Universal Robots PolyScope program: Cinta_1.urp

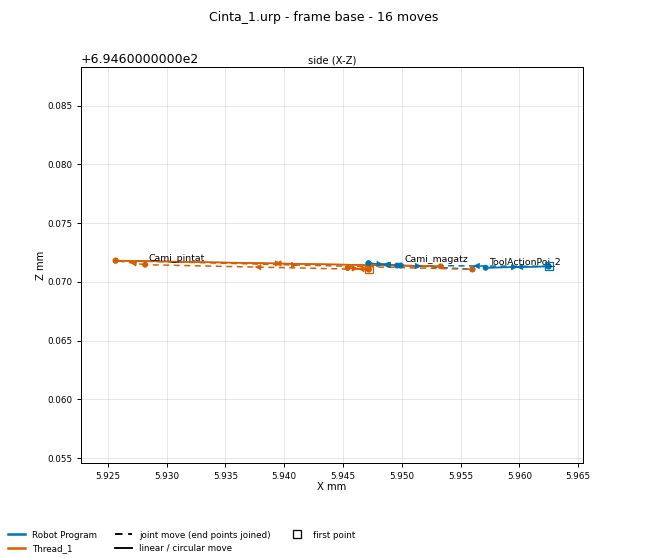
[picture p0: tool path of Cinta_1.urp in frame base, 16 of 16 moves have a stored position in this frame; points joined in program order, loops and branches not executed]
Program Cinta_1 (installation=default directory=/programs createdIn=5.14.5 lastSavedIn=5.14.5 robotSerialNumber=20195300809)
Calibrated DH parameters: a=[-0.000085, -0.20076, -0.212369, 0.000121, -0.000118, 0]; d=[0.15185, -26.306375, 24.753047, 1.684739, 0.085386, 0.092088]; alpha=[1.572149, -0.00522, -0.011864, 1.571339, -1.571085, 0]; deltaTheta=[0, 0.599885, -0.513355, -0.086555, 0.000006, 0]
InitVariablesNode variables(variable(name=Pallet_1_cnt_1, expression=1), variable(name=Pallet_1_lct, expression=1), variable(name=Pallet_1_lno, expression=1), variable(name=Pallet_1_sep, expression=False), variable(name=Pallet_1_tct, expression=1), variable(name=Pallet_2_cnt_1, expression=1), variable(name=Pallet_2_lct, expression=1), variable(name=Pallet_2_lno, expression=1), variable(name=Pallet_2_sep, expression=False), variable(name=Pallet_2_tct, expression=1), variable(name=Pallet_3_cnt, expression=1), variable(name=Pallet_3_lct, expression=1), variable(name=Pallet_3_lno, expression=1), variable(name=Pallet_3_sep, expression=False), variable(name=Pallet_3_tct, expression=1), variable(name=Pallet_4_cnt, expression=1), variable(name=Pallet_4_lct, expression=1), variable(name=Pallet_4_lno, expression=1), variable(name=Pallet_4_sep, expression=False), variable(name=Pallet_4_tct, expression=1))
Robot Program (runOnlyOnce=false)
  If timer_1≟5  and inici≟get_actual_tcp_pose()
    URCap Palletizing (polyscope-pallet-impl, Universal Robots) dataModel(palletFeature=Base, isPalletizing=false, Variable(key=name, variable(name=Pallet_3)), Variable(key=globalCountingVariable, variable(name=Pallet_3_cnt, initializeExpression=1)), Variable(key=layerNumberVariable, variable(name=Pallet_3_lno, initializeExpression=1)), Variable(key=layerCountingVariable, variable(name=Pallet_3_lct, initializeExpression=1)), Variable(key=handleSeparatorVariable, variable(name=Pallet_3_sep, initializeExpression=False)), Variable(key=totalCountVariable, variable(name=Pallet_3_tct, initializeExpression=1)), Length(key=objectHeight value=0.05 unit=M), Variable(key=referencePoint, variable(featureName=referencePoin_2)), Variable(key=separatorPoint, variable(featureName=separatorPoin_2))); state(isChildrenLocked=true)
      URCap Patterns (polyscope-pallet-impl, Universal Robots) state(isChildrenLocked=true)
        URCap Pattern (polyscope-pallet-impl, Universal Robots) dataModel(UUID=57716a2e-ea0b-4b86-9d22-23fb6d1bb1b5, patternType=IRREGULAR, Variable(key=nameVariable, variable(name=Irreg_Pattern_3))); state(isChildrenLocked=true)
          URCap Item (polyscope-pallet-impl, Universal Robots) dataModel(UUID=925eac26-10bc-4873-a4ec-01d33931e9e1, patternType=IRREGULAR, index=0, calibrationDeltaTheta=[2.0871938292282843E-8, 0.5998849625986696, -0.513354759222901, -0.08655474087847535, 6.239817607139875E-6, -6.658617090343766E-8], calibrationA=[-8.52060452638757E-5, -0.2007601879611388, -0.2123691625519033, 1.2105607098011576E-4, -1.1833705743435544E-4, 0.0], calibrationD=[0.15184970286177432, -26.306374840159272, 24.75304670983349, 1.6847390881089916, 0.085385969004481, 0.09208826337351553], calibrationAlpha=[1.5721487795181908, -0.005219907129425837, -0.011864150755780208, 1.5713392161993658, -1.5710853432049288, 0.0], calibrationJointChecksum=[-1860213401, -1859864814, -1494669377, -1328152407, -1329437658, -1329056899], calibrationStatus=2, calibrationValidChecksum=true, baseToFeature=[0.0, 0.0, 0.0, 0.0, 0.0, 0.0], TCPOffset=[-3.816685185402386E-6, 1.2180760577962246E-7, 0.15000008227769798, -3.269188807254424E-7, 6.278455909932198E-6, -1.926188929202367E-5], Variable(key=variable, variable(name=Item_3)), JointPositions(key=jointpositions, JointPosition(key=[1], Angle(key=pos value=0.000066 unit=RAD)), JointPosition(key=[2], Angle(key=pos value=-1.570806 unit=RAD)), JointPosition(key=[3], Angle(key=pos value=0.000024 unit=RAD)), JointPosition(key=[4], Angle(key=pos value=-1.570762 unit=RAD)), JointPosition(key=[5], Angle(key=pos value=-0.000043 unit=RAD)), JointPosition(key=[6], Angle(key=pos value=-0.000104 unit=RAD))))
      URCap Layers (polyscope-pallet-impl, Universal Robots) dataModel(separators=[false], selectedPatterns=[57716a2e-ea0b-4b86-9d22-23fb6d1bb1b5])
      URCap At Each Item (polyscope-pallet-impl, Universal Robots) dataModel(selectedPattern=57716a2e-ea0b-4b86-9d22-23fb6d1bb1b5, selectedPosition=925eac26-10bc-4873-a4ec-01d33931e9e1, Approach_calibrationDeltaTheta=[2.0871938292282843E-8, 0.5998849625986696, -0.513354759222901, -0.08655474087847535, 6.239817607139875E-6, -6.658617090343766E-8], Approach_calibrationA=[-8.52060452638757E-5, -0.2007601879611388, -0.2123691625519033, 1.2105607098011576E-4, -1.1833705743435544E-4, 0.0], Approach_calibrationD=[0.15184970286177432, -26.306374840159272, 24.75304670983349, 1.6847390881089916, 0.085385969004481, 0.09208826337351553], Approach_calibrationAlpha=[1.5721487795181908, -0.005219907129425837, -0.011864150755780208, 1.5713392161993658, -1.5710853432049288, 0.0], Approach_calibrationJointChecksum=[-1860213401, -1859864814, -1494669377, -1328152407, -1329437658, -1329056899], Approach_calibrationStatus=2, Approach_calibrationValidChecksum=true, Approach_baseToFeature=[0.0, 0.0, 0.0, 0.0, 0.0, 0.0], Approach_TCPOffset=[-9.173349571223492E-6, 4.750605908654393E-9, 0.15000004581161422, -1.2312542340189748E-8, -2.3772295653205082E-5, -6.665466225263506E-6], Exit_calibrationDeltaTheta=[2.0871938292282843E-8, 0.5998849625986696, -0.513354759222901, -0.08655474087847535, 6.239817607139875E-6, -6.658617090343766E-8], Exit_calibrationA=[-8.52060452638757E-5, -0.2007601879611388, -0.2123691625519033, 1.2105607098011576E-4, -1.1833705743435544E-4, 0.0], Exit_calibrationD=[0.15184970286177432, -26.306374840159272, 24.75304670983349, 1.6847390881089916, 0.085385969004481, 0.09208826337351553], Exit_calibrationAlpha=[1.5721487795181908, -0.005219907129425837, -0.011864150755780208, 1.5713392161993658, -1.5710853432049288, 0.0], Exit_calibrationJointChecksum=[-1860213401, -1859864814, -1494669377, -1328152407, -1329437658, -1329056899], Exit_calibrationStatus=2, Exit_calibrationValidChecksum=true, Exit_baseToFeature=[0.0, 0.0, 0.0, 0.0, 0.0, 0.0], Exit_TCPOffset=[1.4942311595496577E-5, 5.093315802451315E-8, 0.1500000438837152, -1.396915314811311E-7, 7.536789619608266E-5, -3.90601478415621E-5], currentWizardState=LANDING, Pose(key=refBaseToFeature, Position(key=posePosition, Length(key=X value=0 unit=M), Length(key=Y value=0 unit=M), Length(key=Z value=0 unit=M)), Rotation(key=poseRotation, Angle(key=RX value=0 unit=RAD), Angle(key=RY value=0 unit=RAD), Angle(key=RZ value=0 unit=RAD))), Pose(key=refPose, Position(key=posePosition, Length(key=X value=0.005957 unit=M), Length(key=Y value=-0.3727 unit=M), Length(key=Z value=0.694671 unit=M)), Rotation(key=poseRotation, Angle(key=RX value=-0.017988 unit=RAD), Angle(key=RY value=2.210197 unit=RAD), Angle(key=RZ value=-2.216559 unit=RAD))), JointPositions(key=Approach_jointpositions, JointPosition(key=[1], Angle(key=pos value=0.000066 unit=RAD)), JointPosition(key=[2], Angle(key=pos value=-1.570806 unit=RAD)), JointPosition(key=[3], Angle(key=pos value=0.000024 unit=RAD)), JointPosition(key=[4], Angle(key=pos value=-1.570762 unit=RAD)), JointPosition(key=[5], Angle(key=pos value=-0.000043 unit=RAD)), JointPosition(key=[6], Angle(key=pos value=-0.000104 unit=RAD))), JointPositions(key=Exit_jointpositions, JointPosition(key=[1], Angle(key=pos value=0.000066 unit=RAD)), JointPosition(key=[2], Angle(key=pos value=-1.570806 unit=RAD)), JointPosition(key=[3], Angle(key=pos value=0.000024 unit=RAD)), JointPosition(key=[4], Angle(key=pos value=-1.570762 unit=RAD)), JointPosition(key=[5], Angle(key=pos value=-0.000043 unit=RAD)), JointPosition(key=[6], Angle(key=pos value=-0.000104 unit=RAD))))
        URCap Generated Movements (polyscope-pallet-impl, Universal Robots) state(isChildrenLocked=true)
          MoveJ speed 60 deg/s, acceleration 80 deg/s^2 (useActiveTCP=true) feature=referencePoin_2
            Waypoint Approach_3: TCP in base x=5.962 y=-372.7 z=694.671 mm, rx=-0.018 ry=2.2102 rz=-2.2165 rad; joints [0.004, -90.001, 0.001, -89.998, -0.002, -0.006] deg; TCP offset x=-0.009 y=0 z=150 mm, rx=0 ry=0 rz=0 rad; feature pose in base x=5.957 y=-372.7 z=694.671 mm, rx=-0.018 ry=2.2102 rz=-2.2166 rad
          MoveL speed 250 mm/s, acceleration 1200 mm/s^2 (useActiveTCP=true) feature(featureName=referencePoin_2)
            Waypoint ToolActionPoi_2: TCP in base x=5.957 y=-372.7 z=694.671 mm, rx=-0.018 ry=2.2102 rz=-2.2166 rad; joints [0.004, -90.001, 0.001, -89.998, -0.002, -0.006] deg; TCP offset x=-0.004 y=0 z=150 mm, rx=0 ry=0 rz=0 rad
          Folder Tool action
            URCap Gripper Activate (Robotiq_Grippers, Robotiq Inc.) dataModel(ResetAndActivateKey=false)
            URCap Gripper (Robotiq_Grippers, Robotiq Inc.) dataModel(position=100.0, force=100.0, speed=100.0, positionInDouble=100.0, forceInDouble=100.0, speedInDouble=100.0, slaveIds=[3], blocking=true)
          MoveL speed 250 mm/s, acceleration 1200 mm/s^2 (useActiveTCP=true) feature(featureName=referencePoin_2)
            Waypoint Approach_3: TCP in base x=5.962 y=-372.7 z=694.671 mm, rx=-0.018 ry=2.2102 rz=-2.2165 rad; joints [0.004, -90.001, 0.001, -89.998, -0.002, -0.006] deg; TCP offset x=-0.009 y=0 z=150 mm, rx=0 ry=0 rz=0 rad
    Timer (action=Reset) variable=timer_1
    MoveJ speed 60 deg/s, acceleration 80 deg/s^2 (useActiveTCP=true) feature=Base
      Waypoint Cami_magatz: TCP in base x=5.95 y=-372.7 z=694.671 mm, rx=-0.018 ry=2.2102 rz=-2.2165 rad; joints [0.003, -89.998, -0.001, -89.999, 0, -0.006] deg; TCP offset x=0 y=0 z=150 mm, rx=0 ry=0 rz=0 rad
    URCap Palletizing (polyscope-pallet-impl, Universal Robots) dataModel(palletFeature=Base, isPalletizing=true, Variable(key=name, variable(name=Pallet_4)), Variable(key=globalCountingVariable, variable(name=Pallet_4_cnt, initializeExpression=1)), Variable(key=layerNumberVariable, variable(name=Pallet_4_lno, initializeExpression=1)), Variable(key=layerCountingVariable, variable(name=Pallet_4_lct, initializeExpression=1)), Variable(key=handleSeparatorVariable, variable(name=Pallet_4_sep, initializeExpression=False)), Variable(key=totalCountVariable, variable(name=Pallet_4_tct, initializeExpression=1)), Length(key=objectHeight value=0.05 unit=M), Variable(key=referencePoint, variable(featureName=referencePoin_3)), Variable(key=separatorPoint, variable(featureName=separatorPoin_3))); state(isChildrenLocked=true)
      URCap Patterns (polyscope-pallet-impl, Universal Robots) state(isChildrenLocked=true)
        URCap Pattern (polyscope-pallet-impl, Universal Robots) dataModel(UUID=b4bb1d7d-5fde-484b-989b-01361cd0b8c8, patternType=GRID, columns=3, rows=2, Variable(key=nameVariable, variable(name=Grid_Pattern_1))); state(isChildrenLocked=true)
          URCap Item (polyscope-pallet-impl, Universal Robots) dataModel(UUID=ea4672ff-ad46-4f60-b6cc-b4929b8f2d82, patternType=GRID, index=0, calibrationDeltaTheta=[2.0871938292282843E-8, 0.5998849625986696, -0.513354759222901, -0.08655474087847535, 6.239817607139875E-6, -6.658617090343766E-8], calibrationA=[-8.52060452638757E-5, -0.2007601879611388, -0.2123691625519033, 1.2105607098011576E-4, -1.1833705743435544E-4, 0.0], calibrationD=[0.15184970286177432, -26.306374840159272, 24.75304670983349, 1.6847390881089916, 0.085385969004481, 0.09208826337351553], calibrationAlpha=[1.5721487795181908, -0.005219907129425837, -0.011864150755780208, 1.5713392161993658, -1.5710853432049288, 0.0], calibrationJointChecksum=[-1860213401, -1859864814, -1494669377, -1328152407, -1329437658, -1329056899], calibrationStatus=2, calibrationValidChecksum=true, baseToFeature=[0.0, 0.0, 0.0, 0.0, 0.0, 0.0], TCPOffset=[3.706625326079351E-6, -6.568721999666849E-8, 0.1499998351964846, 1.7803460385569988E-7, -2.84075927765461E-5, 7.288919322566488E-5], Variable(key=variable, variable(name=CornerItem_1)), JointPositions(key=jointpositions, JointPosition(key=[1], Angle(key=pos value=0.000066 unit=RAD)), JointPosition(key=[2], Angle(key=pos value=-1.570806 unit=RAD)), JointPosition(key=[3], Angle(key=pos value=0.000024 unit=RAD)), JointPosition(key=[4], Angle(key=pos value=-1.570762 unit=RAD)), JointPosition(key=[5], Angle(key=pos value=-0.000043 unit=RAD)), JointPosition(key=[6], Angle(key=pos value=-0.000104 unit=RAD))))
          URCap Item (polyscope-pallet-impl, Universal Robots) dataModel(UUID=3c8cbbac-938b-4c56-9b32-ce584113983f, patternType=GRID, index=1, calibrationDeltaTheta=[2.0871938292282843E-8, 0.5998849625986696, -0.513354759222901, -0.08655474087847535, 6.239817607139875E-6, -6.658617090343766E-8], calibrationA=[-8.52060452638757E-5, -0.2007601879611388, -0.2123691625519033, 1.2105607098011576E-4, -1.1833705743435544E-4, 0.0], calibrationD=[0.15184970286177432, -26.306374840159272, 24.75304670983349, 1.6847390881089916, 0.085385969004481, 0.09208826337351553], calibrationAlpha=[1.5721487795181908, -0.005219907129425837, -0.011864150755780208, 1.5713392161993658, -1.5710853432049288, 0.0], calibrationJointChecksum=[-1860213401, -1859864814, -1494669377, -1328152407, -1329437658, -1329056899], calibrationStatus=2, calibrationValidChecksum=true, baseToFeature=[0.0, 0.0, 0.0, 0.0, 0.0, 0.0], TCPOffset=[2.7653235355128386E-6, -9.380526122537702E-8, 0.14999986642115146, 2.5363061092848244E-7, -3.291938284878605E-5, 8.376623252079835E-5], Variable(key=variable, variable(name=CornerItem_2)), JointPositions(key=jointpositions, JointPosition(key=[1], Angle(key=pos value=0.000066 unit=RAD)), JointPosition(key=[2], Angle(key=pos value=-1.570806 unit=RAD)), JointPosition(key=[3], Angle(key=pos value=0.000024 unit=RAD)), JointPosition(key=[4], Angle(key=pos value=-1.570762 unit=RAD)), JointPosition(key=[5], Angle(key=pos value=-0.000043 unit=RAD)), JointPosition(key=[6], Angle(key=pos value=-0.000104 unit=RAD))))
          URCap Item (polyscope-pallet-impl, Universal Robots) dataModel(UUID=2cf3f14a-6e3f-451d-932b-53298661eecf, patternType=GRID, index=2, calibrationDeltaTheta=[2.0871938292282843E-8, 0.5998849625986696, -0.513354759222901, -0.08655474087847535, 6.239817607139875E-6, -6.658617090343766E-8], calibrationA=[-8.52060452638757E-5, -0.2007601879611388, -0.2123691625519033, 1.2105607098011576E-4, -1.1833705743435544E-4, 0.0], calibrationD=[0.15184970286177432, -26.306374840159272, 24.75304670983349, 1.6847390881089916, 0.085385969004481, 0.09208826337351553], calibrationAlpha=[1.5721487795181908, -0.005219907129425837, -0.011864150755780208, 1.5713392161993658, -1.5710853432049288, 0.0], calibrationJointChecksum=[-1860213401, -1859864814, -1494669377, -1328152407, -1329437658, -1329056899], calibrationStatus=2, calibrationValidChecksum=true, baseToFeature=[0.0, 0.0, 0.0, 0.0, 0.0, 0.0], TCPOffset=[6.661449581522492E-6, -2.8157898013247973E-8, 0.14999986386340233, 7.727304519782606E-8, -8.86927201442442E-6, 2.161822139559004E-5], Variable(key=variable, variable(name=CornerItem_3)), JointPositions(key=jointpositions, JointPosition(key=[1], Angle(key=pos value=0.000066 unit=RAD)), JointPosition(key=[2], Angle(key=pos value=-1.570806 unit=RAD)), JointPosition(key=[3], Angle(key=pos value=0.000024 unit=RAD)), JointPosition(key=[4], Angle(key=pos value=-1.570762 unit=RAD)), JointPosition(key=[5], Angle(key=pos value=-0.000043 unit=RAD)), JointPosition(key=[6], Angle(key=pos value=-0.000104 unit=RAD))))
          URCap Item (polyscope-pallet-impl, Universal Robots) dataModel(UUID=14d9bcbf-007f-432e-bf4f-c9794471ffca, patternType=GRID, index=3, calibrationDeltaTheta=[2.0871938292282843E-8, 0.5998849625986696, -0.513354759222901, -0.08655474087847535, 6.239817607139875E-6, -6.658617090343766E-8], calibrationA=[-8.52060452638757E-5, -0.2007601879611388, -0.2123691625519033, 1.2105607098011576E-4, -1.1833705743435544E-4, 0.0], calibrationD=[0.15184970286177432, -26.306374840159272, 24.75304670983349, 1.6847390881089916, 0.085385969004481, 0.09208826337351553], calibrationAlpha=[1.5721487795181908, -0.005219907129425837, -0.011864150755780208, 1.5713392161993658, -1.5710853432049288, 0.0], calibrationJointChecksum=[-1860213401, -1859864814, -1494669377, -1328152407, -1329437658, -1329056899], calibrationStatus=2, calibrationValidChecksum=true, baseToFeature=[0.0, 0.0, 0.0, 0.0, 0.0, 0.0], TCPOffset=[1.0340064511891772E-5, 7.285286818259351E-9, 0.14999993799630948, -1.833199459164639E-8, 1.5011074807964001E-5, 3.57335615816047E-5], Variable(key=variable, variable(name=CornerItem_4)), JointPositions(key=jointpositions, JointPosition(key=[1], Angle(key=pos value=0.000066 unit=RAD)), JointPosition(key=[2], Angle(key=pos value=-1.570806 unit=RAD)), JointPosition(key=[3], Angle(key=pos value=0.000024 unit=RAD)), JointPosition(key=[4], Angle(key=pos value=-1.570762 unit=RAD)), JointPosition(key=[5], Angle(key=pos value=-0.000043 unit=RAD)), JointPosition(key=[6], Angle(key=pos value=-0.000104 unit=RAD))))
      URCap Layers (polyscope-pallet-impl, Universal Robots) dataModel(separators=[false], selectedPatterns=[b4bb1d7d-5fde-484b-989b-01361cd0b8c8])
      URCap At Each Item (polyscope-pallet-impl, Universal Robots) dataModel(selectedPattern=b4bb1d7d-5fde-484b-989b-01361cd0b8c8, selectedPosition=ea4672ff-ad46-4f60-b6cc-b4929b8f2d82, Approach_calibrationDeltaTheta=[2.0871938292282843E-8, 0.5998849625986696, -0.513354759222901, -0.08655474087847535, 6.239817607139875E-6, -6.658617090343766E-8], Approach_calibrationA=[-8.52060452638757E-5, -0.2007601879611388, -0.2123691625519033, 1.2105607098011576E-4, -1.1833705743435544E-4, 0.0], Approach_calibrationD=[0.15184970286177432, -26.306374840159272, 24.75304670983349, 1.6847390881089916, 0.085385969004481, 0.09208826337351553], Approach_calibrationAlpha=[1.5721487795181908, -0.005219907129425837, -0.011864150755780208, 1.5713392161993658, -1.5710853432049288, 0.0], Approach_calibrationJointChecksum=[-1860213401, -1859864814, -1494669377, -1328152407, -1329437658, -1329056899], Approach_calibrationStatus=2, Approach_calibrationValidChecksum=true, Approach_baseToFeature=[0.0, 0.0, 0.0, 0.0, 0.0, 0.0], Approach_TCPOffset=[1.2260157876470355E-5, 1.7997266488212205E-7, 0.15000020897499086, -4.816496149447011E-7, 6.372683936259518E-5, 4.625831555936386E-5], Exit_calibrationDeltaTheta=[2.0871938292282843E-8, 0.5998849625986696, -0.513354759222901, -0.08655474087847535, 6.239817607139875E-6, -6.658617090343766E-8], Exit_calibrationA=[-8.52060452638757E-5, -0.2007601879611388, -0.2123691625519033, 1.2105607098011576E-4, -1.1833705743435544E-4, 0.0], Exit_calibrationD=[0.15184970286177432, -26.306374840159272, 24.75304670983349, 1.6847390881089916, 0.085385969004481, 0.09208826337351553], Exit_calibrationAlpha=[1.5721487795181908, -0.005219907129425837, -0.011864150755780208, 1.5713392161993658, -1.5710853432049288, 0.0], Exit_calibrationJointChecksum=[-1860213401, -1859864814, -1494669377, -1328152407, -1329437658, -1329056899], Exit_calibrationStatus=2, Exit_calibrationValidChecksum=true, Exit_baseToFeature=[0.0, 0.0, 0.0, 0.0, 0.0, 0.0], Exit_TCPOffset=[-1.2169878906291521E-5, -4.481712323478604E-8, 0.14999995430995886, 1.2071276265020752E-7, -4.362424792980929E-5, 4.833778731325504E-6], currentWizardState=LANDING, Pose(key=refBaseToFeature, Position(key=posePosition, Length(key=X value=0 unit=M), Length(key=Y value=0 unit=M), Length(key=Z value=0 unit=M)), Rotation(key=poseRotation, Angle(key=RX value=0 unit=RAD), Angle(key=RY value=0 unit=RAD), Angle(key=RZ value=0 unit=RAD))), Pose(key=refPose, Position(key=posePosition, Length(key=X value=0.00595 unit=M), Length(key=Y value=-0.3727 unit=M), Length(key=Z value=0.694671 unit=M)), Rotation(key=poseRotation, Angle(key=RX value=-0.017924 unit=RAD), Angle(key=RY value=2.210134 unit=RAD), Angle(key=RZ value=-2.216495 unit=RAD))), JointPositions(key=Approach_jointpositions, JointPosition(key=[1], Angle(key=pos value=0.000066 unit=RAD)), JointPosition(key=[2], Angle(key=pos value=-1.570806 unit=RAD)), JointPosition(key=[3], Angle(key=pos value=0.000024 unit=RAD)), JointPosition(key=[4], Angle(key=pos value=-1.570762 unit=RAD)), JointPosition(key=[5], Angle(key=pos value=-0.000043 unit=RAD)), JointPosition(key=[6], Angle(key=pos value=-0.000104 unit=RAD))), JointPositions(key=Exit_jointpositions, JointPosition(key=[1], Angle(key=pos value=0.000066 unit=RAD)), JointPosition(key=[2], Angle(key=pos value=-1.570806 unit=RAD)), JointPosition(key=[3], Angle(key=pos value=0.000024 unit=RAD)), JointPosition(key=[4], Angle(key=pos value=-1.570762 unit=RAD)), JointPosition(key=[5], Angle(key=pos value=-0.000043 unit=RAD)), JointPosition(key=[6], Angle(key=pos value=-0.000104 unit=RAD))))
        URCap Generated Movements (polyscope-pallet-impl, Universal Robots) state(isChildrenLocked=true)
          MoveJ speed 60 deg/s, acceleration 80 deg/s^2 (useActiveTCP=true) feature=referencePoin_3
            Waypoint Approach_4: TCP in base x=5.947 y=-372.7 z=694.672 mm, rx=-0.0179 ry=2.2102 rz=-2.2165 rad; joints [0.006, -89.999, 0.003, -90.002, -0.004, -0.002] deg; feature pose in base x=5.95 y=-372.7 z=694.671 mm, rx=-0.0179 ry=2.2101 rz=-2.2165 rad
          MoveL speed 250 mm/s, acceleration 1200 mm/s^2 (useActiveTCP=true) feature(featureName=referencePoin_3)
            Waypoint ToolActionPoi_3: TCP in base x=5.95 y=-372.7 z=694.671 mm, rx=-0.0179 ry=2.2101 rz=-2.2165 rad; joints [0.004, -90.001, 0.001, -89.998, -0.002, -0.006] deg; TCP offset x=0.004 y=0 z=150 mm, rx=0 ry=0 rz=0.0001 rad
          Folder Tool action
            URCap Gripper (Robotiq_Grippers, Robotiq Inc.) dataModel(position=0.0, force=100.0, speed=100.0, positionInDouble=0.0, forceInDouble=100.0, speedInDouble=100.0, slaveIds=[3], blocking=true)
          MoveL speed 250 mm/s, acceleration 1200 mm/s^2 (useActiveTCP=true) feature(featureName=referencePoin_3)
            Waypoint Approach_4: TCP in base x=5.947 y=-372.7 z=694.672 mm, rx=-0.0179 ry=2.2102 rz=-2.2165 rad; joints [0.006, -89.999, 0.003, -90.002, -0.004, -0.002] deg; TCP offset x=0 y=0 z=150 mm, rx=0 ry=0 rz=0 rad
    Popup Message (haltProgram=false message=Peca al magatzem inputType=Text)
    MoveJ speed 60 deg/s, acceleration 80 deg/s^2 (useActiveTCP=true) feature=Base
      Waypoint inici: TCP in base x=5.956 y=-372.701 z=694.671 mm, rx=-0.0179 ry=2.2102 rz=-2.2166 rad; joints [0.002, -90.002, 0, -89.996, -0.004, -0.005] deg
Thread Thread_1 (runOnlyOnce=false)
  If digital_in[0]≠0  and timer_1≟0  and inici≟get_actual_tcp_pose()
    URCap Palletizing (polyscope-pallet-impl, Universal Robots) dataModel(palletFeature=Base, isPalletizing=true, Variable(key=name, variable(name=Pallet_1)), Variable(key=globalCountingVariable, variable(name=Pallet_1_cnt_1, initializeExpression=1)), Variable(key=layerNumberVariable, variable(name=Pallet_1_lno, initializeExpression=1)), Variable(key=layerCountingVariable, variable(name=Pallet_1_lct, initializeExpression=1)), Variable(key=handleSeparatorVariable, variable(name=Pallet_1_sep, initializeExpression=False)), Variable(key=totalCountVariable, variable(name=Pallet_1_tct, initializeExpression=1)), Length(key=objectHeight value=0.05 unit=M), Variable(key=referencePoint, variable(featureName=referencePoint)), Variable(key=separatorPoint, variable(featureName=separatorPoint))); state(isChildrenLocked=true)
      URCap Patterns (polyscope-pallet-impl, Universal Robots) state(isChildrenLocked=true)
        URCap Pattern (polyscope-pallet-impl, Universal Robots) dataModel(UUID=fc05b72d-a196-495d-97c6-d9a1d159b760, patternType=IRREGULAR, Variable(key=nameVariable, variable(name=Irreg_Pattern_1))); state(isChildrenLocked=true)
          URCap Item (polyscope-pallet-impl, Universal Robots) dataModel(UUID=fe7b0d55-38a9-456e-bd41-5611c4695fc9, patternType=IRREGULAR, index=0, calibrationDeltaTheta=[2.0871938292282843E-8, 0.5998849625986696, -0.513354759222901, -0.08655474087847535, 6.239817607139875E-6, -6.658617090343766E-8], calibrationA=[-8.52060452638757E-5, -0.2007601879611388, -0.2123691625519033, 1.2105607098011576E-4, -1.1833705743435544E-4, 0.0], calibrationD=[0.15184970286177432, -26.306374840159272, 24.75304670983349, 1.6847390881089916, 0.085385969004481, 0.09208826337351553], calibrationAlpha=[1.5721487795181908, -0.005219907129425837, -0.011864150755780208, 1.5713392161993658, -1.5710853432049288, 0.0], calibrationJointChecksum=[-1860213401, -1859864814, -1494669377, -1328152407, -1329437658, -1329056899], calibrationStatus=2, calibrationValidChecksum=true, baseToFeature=[0.0, 0.0, 0.0, 0.0, 0.0, 0.0], TCPOffset=[-1.751886057855509E-6, 1.0215014467629402E-7, 0.15000017116993, -2.7439439849184956E-7, 2.951747630344638E-5, -7.270362872304238E-5], Variable(key=variable, variable(name=Item_1)), JointPositions(key=jointpositions, JointPosition(key=[1], Angle(key=pos value=0 unit=RAD)), JointPosition(key=[2], Angle(key=pos value=-1.570796 unit=RAD)), JointPosition(key=[3], Angle(key=pos value=0 unit=RAD)), JointPosition(key=[4], Angle(key=pos value=-1.570796 unit=RAD)), JointPosition(key=[5], Angle(key=pos value=0 unit=RAD)), JointPosition(key=[6], Angle(key=pos value=0 unit=RAD))))
      URCap Layers (polyscope-pallet-impl, Universal Robots) dataModel(separators=[false], selectedPatterns=[fc05b72d-a196-495d-97c6-d9a1d159b760])
      URCap At Each Item (polyscope-pallet-impl, Universal Robots) dataModel(selectedPattern=fc05b72d-a196-495d-97c6-d9a1d159b760, selectedPosition=fe7b0d55-38a9-456e-bd41-5611c4695fc9, Approach_calibrationDeltaTheta=[2.0871938292282843E-8, 0.5998849625986696, -0.513354759222901, -0.08655474087847535, 6.239817607139875E-6, -6.658617090343766E-8], Approach_calibrationA=[-8.52060452638757E-5, -0.2007601879611388, -0.2123691625519033, 1.2105607098011576E-4, -1.1833705743435544E-4, 0.0], Approach_calibrationD=[0.15184970286177432, -26.306374840159272, 24.75304670983349, 1.6847390881089916, 0.085385969004481, 0.09208826337351553], Approach_calibrationAlpha=[1.5721487795181908, -0.005219907129425837, -0.011864150755780208, 1.5713392161993658, -1.5710853432049288, 0.0], Approach_calibrationJointChecksum=[-1860213401, -1859864814, -1494669377, -1328152407, -1329437658, -1329056899], Approach_calibrationStatus=2, Approach_calibrationValidChecksum=true, Approach_baseToFeature=[0.0, 0.0, 0.0, 0.0, 0.0, 0.0], Approach_TCPOffset=[-3.5489445641637563E-6, 2.2419070278001385E-7, 0.1500002388481764, -6.002459325721902E-7, 4.246931429269476E-5, -5.3457643173503646E-5], Exit_calibrationDeltaTheta=[2.0871938292282843E-8, 0.5998849625986696, -0.513354759222901, -0.08655474087847535, 6.239817607139875E-6, -6.658617090343766E-8], Exit_calibrationA=[-8.52060452638757E-5, -0.2007601879611388, -0.2123691625519033, 1.2105607098011576E-4, -1.1833705743435544E-4, 0.0], Exit_calibrationD=[0.15184970286177432, -26.306374840159272, 24.75304670983349, 1.6847390881089916, 0.085385969004481, 0.09208826337351553], Exit_calibrationAlpha=[1.5721487795181908, -0.005219907129425837, -0.011864150755780208, 1.5713392161993658, -1.5710853432049288, 0.0], Exit_calibrationJointChecksum=[-1860213401, -1859864814, -1494669377, -1328152407, -1329437658, -1329056899], Exit_calibrationStatus=2, Exit_calibrationValidChecksum=true, Exit_baseToFeature=[0.0, 0.0, 0.0, 0.0, 0.0, 0.0], Exit_TCPOffset=[1.0345607790528501E-6, -1.386905819078521E-7, 0.14999980087328915, 3.723825514563124E-7, -4.3806556485191505E-5, 6.004798123714267E-6], currentWizardState=SHOW_DONE, Pose(key=refBaseToFeature, Position(key=posePosition, Length(key=X value=0 unit=M), Length(key=Y value=0 unit=M), Length(key=Z value=0 unit=M)), Rotation(key=poseRotation, Angle(key=RX value=0 unit=RAD), Angle(key=RY value=0 unit=RAD), Angle(key=RZ value=0 unit=RAD))), Pose(key=refPose, Position(key=posePosition, Length(key=X value=0.005945 unit=M), Length(key=Y value=-0.372701 unit=M), Length(key=Z value=0.694671 unit=M)), Rotation(key=poseRotation, Angle(key=RX value=-0.017934 unit=RAD), Angle(key=RY value=2.210219 unit=RAD), Angle(key=RZ value=-2.216581 unit=RAD))), JointPositions(key=Approach_jointpositions, JointPosition(key=[1], Angle(key=pos value=0 unit=RAD)), JointPosition(key=[2], Angle(key=pos value=-1.570796 unit=RAD)), JointPosition(key=[3], Angle(key=pos value=0 unit=RAD)), JointPosition(key=[4], Angle(key=pos value=-1.570796 unit=RAD)), JointPosition(key=[5], Angle(key=pos value=0 unit=RAD)), JointPosition(key=[6], Angle(key=pos value=0 unit=RAD))), JointPositions(key=Exit_jointpositions, JointPosition(key=[1], Angle(key=pos value=0 unit=RAD)), JointPosition(key=[2], Angle(key=pos value=-1.570796 unit=RAD)), JointPosition(key=[3], Angle(key=pos value=0 unit=RAD)), JointPosition(key=[4], Angle(key=pos value=-1.570796 unit=RAD)), JointPosition(key=[5], Angle(key=pos value=0 unit=RAD)), JointPosition(key=[6], Angle(key=pos value=0 unit=RAD))))
        URCap Generated Movements (polyscope-pallet-impl, Universal Robots) state(isChildrenLocked=true)
          MoveJ speed 60 deg/s, acceleration 80 deg/s^2 (useActiveTCP=true) feature=referencePoint
            Waypoint Approach: TCP in base x=5.947 y=-372.701 z=694.671 mm, rx=-0.0179 ry=2.2102 rz=-2.2166 rad; joints [0, -90, 0, -90, 0, 0] deg; TCP offset x=-0.004 y=0 z=150 mm, rx=0 ry=0 rz=-0.0001 rad; feature pose in base x=5.945 y=-372.701 z=694.671 mm, rx=-0.0179 ry=2.2102 rz=-2.2166 rad
          MoveL speed 250 mm/s, acceleration 1200 mm/s^2 (useActiveTCP=true) feature(featureName=referencePoint)
            Waypoint ToolActionPoint: TCP in base x=5.945 y=-372.701 z=694.671 mm, rx=-0.0179 ry=2.2102 rz=-2.2166 rad; joints [0, -90, 0, -90, 0, 0] deg; TCP offset x=-0.002 y=0 z=150 mm, rx=0 ry=0 rz=-0.0001 rad
          Folder Tool action
            URCap Gripper Activate (Robotiq_Grippers, Robotiq Inc.) dataModel(ResetAndActivateKey=false)
          MoveL speed 250 mm/s, acceleration 1200 mm/s^2 (useActiveTCP=true) feature(featureName=referencePoint)
            Waypoint Approach: TCP in base x=5.947 y=-372.701 z=694.671 mm, rx=-0.0179 ry=2.2102 rz=-2.2166 rad; joints [0, -90, 0, -90, 0, 0] deg; TCP offset x=-0.004 y=0 z=150 mm, rx=0 ry=0 rz=-0.0001 rad
    Popup Message (haltProgram=false message=Object agafat inputType=Text)
    MoveJ speed 60 deg/s, acceleration 80 deg/s^2 (useActiveTCP=true) feature=Base
      Waypoint Cami_pintat: TCP in base x=5.928 y=-372.701 z=694.671 mm, rx=-0.0178 ry=2.2102 rz=-2.2165 rad; joints [0, -90, 0.002, -90.001, -0.001, -0.001] deg; TCP offset x=0 y=0 z=150 mm, rx=0 ry=0 rz=0 rad
    URCap Palletizing (polyscope-pallet-impl, Universal Robots) dataModel(palletFeature=Base, isPalletizing=true, Variable(key=name, variable(name=Pallet_2)), Variable(key=globalCountingVariable, variable(name=Pallet_2_cnt_1, initializeExpression=1)), Variable(key=layerNumberVariable, variable(name=Pallet_2_lno, initializeExpression=1)), Variable(key=layerCountingVariable, variable(name=Pallet_2_lct, initializeExpression=1)), Variable(key=handleSeparatorVariable, variable(name=Pallet_2_sep, initializeExpression=False)), Variable(key=totalCountVariable, variable(name=Pallet_2_tct, initializeExpression=1)), Length(key=objectHeight value=0.05 unit=M), Variable(key=referencePoint, variable(featureName=referencePoin_1)), Variable(key=separatorPoint, variable(featureName=separatorPoin_1))); state(isChildrenLocked=true)
      URCap Patterns (polyscope-pallet-impl, Universal Robots) state(isChildrenLocked=true)
        URCap Pattern (polyscope-pallet-impl, Universal Robots) dataModel(UUID=e3a95b3b-049c-434c-81ef-e175da3fd9c2, patternType=IRREGULAR, Variable(key=nameVariable, variable(name=Irreg_Pattern_2))); state(isChildrenLocked=true)
          URCap Item (polyscope-pallet-impl, Universal Robots) dataModel(UUID=6651543a-c84f-4d9c-8dd1-934f5d3b7aa1, patternType=IRREGULAR, index=0, calibrationDeltaTheta=[2.0871938292282843E-8, 0.5998849625986696, -0.513354759222901, -0.08655474087847535, 6.239817607139875E-6, -6.658617090343766E-8], calibrationA=[-8.52060452638757E-5, -0.2007601879611388, -0.2123691625519033, 1.2105607098011576E-4, -1.1833705743435544E-4, 0.0], calibrationD=[0.15184970286177432, -26.306374840159272, 24.75304670983349, 1.6847390881089916, 0.085385969004481, 0.09208826337351553], calibrationAlpha=[1.5721487795181908, -0.005219907129425837, -0.011864150755780208, 1.5713392161993658, -1.5710853432049288, 0.0], calibrationJointChecksum=[-1860213401, -1859864814, -1494669377, -1328152407, -1329437658, -1329056899], calibrationStatus=2, calibrationValidChecksum=true, baseToFeature=[0.0, 0.0, 0.0, 0.0, 0.0, 0.0], TCPOffset=[-9.672812069199766E-6, -4.48190197177567E-8, 0.150000013883362, 1.2072611746856745E-7, -2.3173632993324257E-5, -5.582307446309488E-5], Variable(key=variable, variable(name=Item_2)), JointPositions(key=jointpositions, JointPosition(key=[1], Angle(key=pos value=0 unit=RAD)), JointPosition(key=[2], Angle(key=pos value=-1.570796 unit=RAD)), JointPosition(key=[3], Angle(key=pos value=0 unit=RAD)), JointPosition(key=[4], Angle(key=pos value=-1.570796 unit=RAD)), JointPosition(key=[5], Angle(key=pos value=0 unit=RAD)), JointPosition(key=[6], Angle(key=pos value=0 unit=RAD))))
      URCap Layers (polyscope-pallet-impl, Universal Robots) dataModel(separators=[false], selectedPatterns=[e3a95b3b-049c-434c-81ef-e175da3fd9c2])
      URCap At Each Item (polyscope-pallet-impl, Universal Robots) dataModel(selectedPattern=e3a95b3b-049c-434c-81ef-e175da3fd9c2, selectedPosition=6651543a-c84f-4d9c-8dd1-934f5d3b7aa1, Approach_calibrationDeltaTheta=[2.0871938292282843E-8, 0.5998849625986696, -0.513354759222901, -0.08655474087847535, 6.239817607139875E-6, -6.658617090343766E-8], Approach_calibrationA=[-8.52060452638757E-5, -0.2007601879611388, -0.2123691625519033, 1.2105607098011576E-4, -1.1833705743435544E-4, 0.0], Approach_calibrationD=[0.15184970286177432, -26.306374840159272, 24.75304670983349, 1.6847390881089916, 0.085385969004481, 0.09208826337351553], Approach_calibrationAlpha=[1.5721487795181908, -0.005219907129425837, -0.011864150755780208, 1.5713392161993658, -1.5710853432049288, 0.0], Approach_calibrationJointChecksum=[-1860213401, -1859864814, -1494669377, -1328152407, -1329437658, -1329056899], Approach_calibrationStatus=2, Approach_calibrationValidChecksum=true, Approach_baseToFeature=[0.0, 0.0, 0.0, 0.0, 0.0, 0.0], Approach_TCPOffset=[4.4697166960552625E-5, -2.960722850220421E-7, 0.14999968340059391, 7.984353551316673E-7, 6.140025800733009E-5, 4.3967758798923496E-5], Exit_calibrationDeltaTheta=[2.0871938292282843E-8, 0.5998849625986696, -0.513354759222901, -0.08655474087847535, 6.239817607139875E-6, -6.658617090343766E-8], Exit_calibrationA=[-8.52060452638757E-5, -0.2007601879611388, -0.2123691625519033, 1.2105607098011576E-4, -1.1833705743435544E-4, 0.0], Exit_calibrationD=[0.15184970286177432, -26.306374840159272, 24.75304670983349, 1.6847390881089916, 0.085385969004481, 0.09208826337351553], Exit_calibrationAlpha=[1.5721487795181908, -0.005219907129425837, -0.011864150755780208, 1.5713392161993658, -1.5710853432049288, 0.0], Exit_calibrationJointChecksum=[-1860213401, -1859864814, -1494669377, -1328152407, -1329437658, -1329056899], Exit_calibrationStatus=2, Exit_calibrationValidChecksum=true, Exit_baseToFeature=[0.0, 0.0, 0.0, 0.0, 0.0, 0.0], Exit_TCPOffset=[3.766030330380814E-5, -4.069868282385869E-7, 0.1499994672907212, 1.0971591498703011E-6, 1.417921471940936E-5, 4.2079585011064136E-5], currentWizardState=LANDING, Pose(key=refBaseToFeature, Position(key=posePosition, Length(key=X value=0 unit=M), Length(key=Y value=0 unit=M), Length(key=Z value=0 unit=M)), Rotation(key=poseRotation, Angle(key=RX value=0 unit=RAD), Angle(key=RY value=0 unit=RAD), Angle(key=RZ value=0 unit=RAD))), Pose(key=refPose, Position(key=posePosition, Length(key=X value=0.005953 unit=M), Length(key=Y value=-0.3727 unit=M), Length(key=Z value=0.694671 unit=M)), Rotation(key=poseRotation, Angle(key=RX value=-0.017973 unit=RAD), Angle(key=RY value=2.210184 unit=RAD), Angle(key=RZ value=-2.216546 unit=RAD))), JointPositions(key=Approach_jointpositions, JointPosition(key=[1], Angle(key=pos value=0.000066 unit=RAD)), JointPosition(key=[2], Angle(key=pos value=-1.570806 unit=RAD)), JointPosition(key=[3], Angle(key=pos value=0.000024 unit=RAD)), JointPosition(key=[4], Angle(key=pos value=-1.570762 unit=RAD)), JointPosition(key=[5], Angle(key=pos value=-0.000043 unit=RAD)), JointPosition(key=[6], Angle(key=pos value=-0.000104 unit=RAD))), JointPositions(key=Exit_jointpositions, JointPosition(key=[1], Angle(key=pos value=0.000066 unit=RAD)), JointPosition(key=[2], Angle(key=pos value=-1.570806 unit=RAD)), JointPosition(key=[3], Angle(key=pos value=0.000024 unit=RAD)), JointPosition(key=[4], Angle(key=pos value=-1.570762 unit=RAD)), JointPosition(key=[5], Angle(key=pos value=-0.000043 unit=RAD)), JointPosition(key=[6], Angle(key=pos value=-0.000104 unit=RAD))))
        URCap Generated Movements (polyscope-pallet-impl, Universal Robots) state(isChildrenLocked=true)
          MoveJ speed 60 deg/s, acceleration 80 deg/s^2 (useActiveTCP=true) feature=referencePoin_1
            Waypoint Approach_2: TCP in base x=5.926 y=-372.7 z=694.672 mm, rx=-0.0179 ry=2.2101 rz=-2.2165 rad; joints [0.006, -89.997, 0.003, -89.998, -0.002, -0.005] deg; feature pose in base x=5.953 y=-372.7 z=694.671 mm, rx=-0.018 ry=2.2102 rz=-2.2165 rad
          MoveL speed 250 mm/s, acceleration 1200 mm/s^2 (useActiveTCP=true) feature(featureName=referencePoin_1)
            Waypoint ToolActionPoi_1: TCP in base x=5.953 y=-372.7 z=694.671 mm, rx=-0.018 ry=2.2102 rz=-2.2165 rad; joints [0, -90, 0, -90, 0, 0] deg; TCP offset x=-0.01 y=0 z=150 mm, rx=0 ry=0 rz=-0.0001 rad
          Folder Tool action
            URCap Gripper (Robotiq_Grippers, Robotiq Inc.) dataModel(position=0.0, force=100.0, speed=100.0, positionInDouble=0.0, forceInDouble=100.0, speedInDouble=100.0, slaveIds=[3], blocking=true)
          MoveL speed 250 mm/s, acceleration 1200 mm/s^2 (useActiveTCP=true) feature(featureName=referencePoin_1)
            Waypoint Approach_2: TCP in base x=5.926 y=-372.7 z=694.672 mm, rx=-0.0179 ry=2.2101 rz=-2.2165 rad; joints [0.006, -89.997, 0.003, -89.998, -0.002, -0.005] deg; TCP offset x=0 y=0 z=150 mm, rx=0 ry=0 rz=0 rad
    Popup Message (haltProgram=false message=pieza pintando inputType=Text)
    MoveJ speed 60 deg/s, acceleration 80 deg/s^2 (useActiveTCP=true) feature=Base
      Waypoint inici referenceName=inici: TCP in base x=5.956 y=-372.701 z=694.671 mm, rx=-0.0179 ry=2.2102 rz=-2.2166 rad; joints [0.002, -90.002, 0, -89.996, -0.004, -0.005] deg
